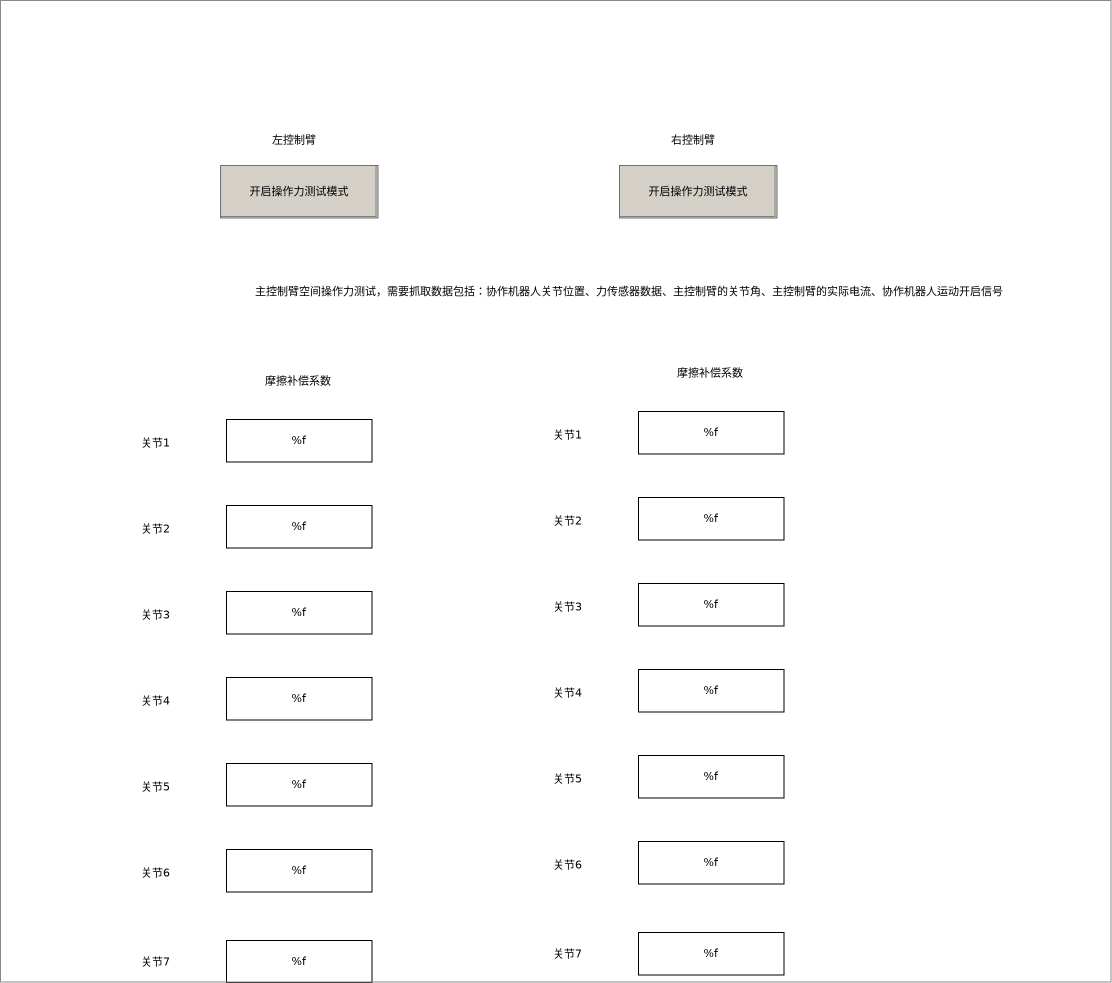
VISUALIZATION manipulateTest  // 1112x983
    Button (220,165 158x53), "开启操作力测试模式", colour toggle: g_maniTest.m_testStart[1]
        toggle g_maniTest.m_testStart[1]
    Label (219,125 150x30), "左控制臂"
    Button (619,165 158x53), "开启操作力测试模式", colour toggle: g_maniTest.m_testStart[2]
        toggle g_maniTest.m_testStart[2]
    Label (618,125 150x30), "右控制臂"
    Label (146,247 966x89), "主控制臂空间操作力测试，需要抓取数据包括：协作机器人关节位置、力传感器数据、主控制臂的关节角、主控制臂的实际电流、协作机器人运动开启信号"
    Rectangle (226,419 146x43), "%f", text variable: g_maniTest.m_frictionFactor[1][1]
        OnMouseClick: write the text variable via Default
    Label (104,425 103x36), "关节1"
    Label (223,366 150x30), "摩擦补偿系数"
    Rectangle (226,505 146x43), "%f", text variable: g_maniTest.m_frictionFactor[1][2]
        OnMouseClick: write the text variable via Default
    Rectangle (226,591 146x43), "%f", text variable: g_maniTest.m_frictionFactor[1][3]
        OnMouseClick: write the text variable via Default
    Rectangle (226,677 146x43), "%f", text variable: g_maniTest.m_frictionFactor[1][4]
        OnMouseClick: write the text variable via Default
    Rectangle (226,763 146x43), "%f", text variable: g_maniTest.m_frictionFactor[1][5]
        OnMouseClick: write the text variable via Default
    Rectangle (226,849 146x43), "%f", text variable: g_maniTest.m_frictionFactor[1][6]
        OnMouseClick: write the text variable via Default
    Rectangle (226,940 146x43), "%f", text variable: g_maniTest.m_frictionFactor[1][7]
        OnMouseClick: write the text variable via Default
    Label (104,511 103x36), "关节2"
    Label (104,597 103x36), "关节3"
    Label (104,683 103x36), "关节4"
    Label (104,769 103x36), "关节5"
    Label (104,855 103x36), "关节6"
    Label (104,944 103x36), "关节7"
    Rectangle (638,411 146x43), "%f", text variable: g_maniTest.m_frictionFactor[2][1]
        OnMouseClick: write the text variable via Default
    Label (516,417 103x36), "关节1"
    Label (635,358 150x30), "摩擦补偿系数"
    Rectangle (638,497 146x43), "%f", text variable: g_maniTest.m_frictionFactor[2][2]
        OnMouseClick: write the text variable via Default
    Rectangle (638,583 146x43), "%f", text variable: g_maniTest.m_frictionFactor[2][3]
        OnMouseClick: write the text variable via Default
    Rectangle (638,669 146x43), "%f", text variable: g_maniTest.m_frictionFactor[2][4]
        OnMouseClick: write the text variable via Default
    Rectangle (638,755 146x43), "%f", text variable: g_maniTest.m_frictionFactor[2][5]
        OnMouseClick: write the text variable via Default
    Rectangle (638,841 146x43), "%f", text variable: g_maniTest.m_frictionFactor[2][6]
        OnMouseClick: write the text variable via Default
    Rectangle (638,932 146x43), "%f", text variable: g_maniTest.m_frictionFactor[2][7]
        OnMouseClick: write the text variable via Default
    Label (516,503 103x36), "关节2"
    Label (516,589 103x36), "关节3"
    Label (516,675 103x36), "关节4"
    Label (516,761 103x36), "关节5"
    Label (516,847 103x36), "关节6"
    Label (516,936 103x36), "关节7"
END_VISUALIZATION

(* stored: Version 1.1.0.1, ProductVersion 3.1.4024.11
   Visu manipulateTest: Id {77acdd2f-bb6b-48a4-834c-74696bdae2f6} *)
